{attribute addProperty BoxType "EPP5101-0002-0016"}
{attribute addProperty Id "ENC_Status_compactAT %I*ENC_Status_compact_18E0726F4860ENC_Control_compactAT %Q*ENC_Control_compact_3146A3B23240WcStateAT %I*WcState_98A4DF7520.250InfoDataAT %I*InfoData_BC63D37F80100"}
{attribute addProperty CRC "3145072827"}
{attribute addProperty SizeInBites "162"}
{attribute addProperty SizeInBytes "20.25"}
TYPE EPP5101_CA84C7C4 :
STRUCT
	{attribute addProperty Name "ENC_Status_compact"}
	ENC_Status_compact : ENC_Status_compact_18E0726F;
	{attribute addProperty Name "ENC_Control_compact"}
	ENC_Control_compact : ENC_Control_compact_3146A3B2;
	{attribute addProperty Name "WcState"}
	WcState : WcState_98A4DF75;
	{attribute addProperty Name "InfoData"}
	InfoData : InfoData_BC63D37F;
END_STRUCT
END_TYPE

(* stored: Version 1.2.0.0, ProductVersion 3.1.4024.9
   DUT EPP5101_CA84C7C4: Id {272f8f72-e152-4d00-b76b-26518519f3a8} *)
